// TIA Portal V16 export
// export: Created 2020-03-17T19:14:23.6206523Z, ExportSetting None, DisplayName Totally Integrated Automation Portal, DisplayVersion V16, DisplayName TIA Portal Version Control Interface, DisplayVersion V16, DisplayName TIA Portal Openness, DisplayVersion V16, DisplayName STEP 7 Professional, DisplayVersion V16, DisplayName STEP 7 Safety, DisplayVersion V16, DisplayName WinCC Advanced, DisplayVersion V16
TYPE "StepValues"
   STRUCT
      StepMode : Int;   // 0 = Automatic / 1 = SingleStep
      SingleStep : Bool;   // Step once
      CurrentStep : Int;   // Actual step no
      CurrentTime : DInt;   // Actual step time
      CylcleState : Int;   // 1 = running
      CycleAbort : Bool;   // abort cycle
   END_STRUCT;
END_TYPE
